{attribute 'qualified_only'}
VAR_GLOBAL CONSTANT
	INDEX_MIN : INT := 1;
	INDEX_MAX : INT := 10;
END_VAR

(* stored: Version 1.1.0.1
   GVL GVL: Id {13a74d90-f2ce-438b-82ed-d2a8506c2e15} *)
